{attribute 'qualified_only'}
{attribute 'strict'}
TYPE E_FT :
(
	PUMP,
	
	CYL1_E,
	CYL1_R,
	CYL2_E,
	CYL2_R,
	CYL3_E,
	CYL3_R,
	CYL4_E,
	CYL4_R,
	CYL5_E,
	CYL5_R,
	CYL6_E,
	CYL6_R,
	CYL7_E,
	CYL7_R,
	
	PCYL1_E,
	PCYL1_R,
	PCYL2_E,
	PCYL2_R
);
END_TYPE

(* stored: Version 1.1.0.1, ProductVersion 3.1.4024.6
   EnumerationTextList E_FT: Id {7cd59841-7c09-48ec-a230-d868594b33a9} *)
